METHOD PROTECTED OnStart
IF NOT Tco_TO_Tc2MC2_HomingMode(_homingMode, _mc_homingMode) THEN
    _message := Tc2_Standard.CONCAT('Unable to cast _homingMode variable of type TcoDrivesBeckhoff.eHomingMode (', TO_STRING(_homingMode));
    _message := Tc2_Standard.CONCAT(_message, ') to the type Tc2_MC2.MC_HomingMode!!!');
    THIS^.Messenger.Post(_message, TcoCore.eMessageCategory.ProgrammingError);
    ThrowWhen(TRUE);
    RETURN;
END_IF

IF NOT Tco_TO_Tc2MC2_Direction(_homingOptions_SearchDirection, _mc_homingOptions_SyncDirection) THEN
    _message := Tc2_Standard.CONCAT('Unable to cast _homingOptions_SearchDirection variable of type TcoDrivesBeckhoff.eDirection (',
        TO_STRING(_homingOptions_SearchDirection));

    _message := Tc2_Standard.CONCAT(_message, ') to the type Tc2_MC2.MC_Direction!!!');
    THIS^.Messenger.Post(_message, TcoCore.eMessageCategory.ProgrammingError);
    ThrowWhen(TRUE);
    RETURN;
END_IF

IF NOT Tco_TO_Tc2MC2_Direction(_homingOptions_SyncDirection, _mc_homingOptions_SyncDirection) THEN
    _message := Tc2_Standard.CONCAT('Unable to cast _homingOptions_SearchDirection variable of type TcoDrivesBeckhoff.eDirection (',
        TO_STRING(_homingOptions_SyncDirection));

    _message := Tc2_Standard.CONCAT(_message, ') to the type Tc2_MC2.MC_Direction!!!');
    THIS^.Messenger.Post(_message, TcoCore.eMessageCategory.ProgrammingError);
    ThrowWhen(TRUE);
    RETURN;
END_IF

IF NOT Tco_TO_Tc2MC2_EncRefMode(_homingOptions_ReferenceMode, _mc_homingOptions_ReferenceMode) THEN
    _message := Tc2_Standard.CONCAT('Unable to cast _homingOptions_ReferenceMode variable of type TcoDrivesBeckhoff.eEncoderReferenceMode (',
        TO_STRING(_homingOptions_ReferenceMode));

    _message := Tc2_Standard.CONCAT(_message, ') to the type Tc2_MC2.E_EncoderReferenceMode!!!');
    THIS^.Messenger.Post(_message, TcoCore.eMessageCategory.ProgrammingError);
    ThrowWhen(TRUE);
    RETURN;
END_IF

_mc_homingOptions.ClearPositionLag := _homingOptions_ClearPositionLag;
_mc_homingOptions.SearchDirection := _homingOptions_SearchDirection;
_mc_homingOptions.SearchVelocity := _homingOptions_SearchVelocity;
_mc_homingOptions.SyncDirection := _homingOptions_SyncDirection;
_mc_homingOptions.SyncVelocity := _homingOptions_SyncVelocity;
_mc_homingOptions.ReferenceMode := _homingOptions_ReferenceMode;
_calibrationCam := DriveRef.inCalibrationCam;
_mcHome(Axis := _axisRef, Execute := FALSE);
END_METHOD

(*~
    <docu>
        <summary>
            Restores this instance to the Ready state. Can be called explicitly or from within one of the restore mechanisms.
            <para>
                See also <see cref="PlcDocu.TcoCore.TcoTask.AutoRestorable()"/>
            </para>
        </summary>
    </docu>
~*)
METHOD Restore : ITcoRestorable
SUPER^.Restore();
END_METHOD

(*~
    <docu>
        <summary>
            Executes until task is in ```Error``` state .
        </summary>
    </docu>
~*)
METHOD PROTECTED WhileError
IF NOT _axisRef.Status.Error THEN
    DriveRef.SetErrorID(DriveRef._homeTask._mcHome.ErrorID);
    _mcHome(Axis := _axisRef, Execute := FALSE);
END_IF
END_METHOD

END_FUNCTION_BLOCK

// ---- POUs/Prototypes/TcoDriveSimple/Jog.TcPOU
FUNCTION_BLOCK Jog EXTENDS TcoCore.TcoObject IMPLEMENTS ITcoDriveSimple, TcoCore.ITcoServiceable
VAR_INPUT
    inIsServiceMode : BOOL;
END_VAR
VAR
    {attribute 'hide'}
    _axisRef : REFERENCE TO TcoAxisRef;
    {attribute 'hide'}
    _mcJog : Tc2_MC2.MC_Jog;
    {attribute addProperty Name "<#Jog forward#>"}
    {attribute addProperty StateOnDesc "<#Running#>"}
    {attribute addProperty StateOffDesc "<#Stopped#>"}
    _jogForwardTask : TcoCore.TcoMomentaryTask(THIS^);
    {attribute addProperty Name "<#Jog backwards#>"}
    {attribute addProperty StateOnDesc "<#Running#>"}
    {attribute addProperty StateOffDesc "<#Stopped#>"}
    _jogBackwardsTask : TcoCore.TcoMomentaryTask(THIS^);
    {attribute addProperty Name "<#Jog mode#>"}
    _jogMode : eJogMode;
    {attribute addProperty Name "<#Position#>"}
    _position : LREAL;
    {attribute addProperty Name "<#Velocity#>"}
    _velocity : LREAL;
    {attribute addProperty Name "<#Acceleration#>"}
    _acceleration : LREAL;
    {attribute addProperty Name "<#Deceleration#>"}
    _deceleration : LREAL;
    {attribute addProperty Name "<#Jerk#>"}
    _jerk : LREAL;
    {attribute 'hide'}
    _dummyPreconditionOK : BOOL;
    _serviceContexCycle : ULINT;
    _myContextCycleCount : ULINT;
    _inServiceMode : BOOL;
END_VAR

IF NOT __ISVALIDREF(_axisRef) THEN
    IF __ISVALIDREF(DriveRef) THEN
        _axisRef REF= DriveRef.AxisRef;
    ELSE
        RETURN;
    END_IF
END_IF

_jogForwardTask.Enabled := inIsServiceMode;
_jogBackwardsTask.Enabled := inIsServiceMode;
_jogForwardTask.Run();
_jogBackwardsTask.Run();

IF _jogForwardTask.State THEN
    _dummyPreconditionOK := DriveRef._power._mcPower.Enable_Positive;

    IF NOT DriveRef._movementState.JogPreconditionsOk(_jogForwardTask, _dummyPreconditionOK) THEN
        Messenger.Error('Movements to positive direction are disabled');
        RETURN;
    END_IF
END_IF

IF _jogBackwardsTask.State THEN
    _dummyPreconditionOK := DriveRef._power._mcPower.Enable_Negative;

    IF NOT DriveRef._movementState.JogPreconditionsOk(_jogBackwardsTask, _dummyPreconditionOK) THEN
        Messenger.Error('Movements to negative direction are disabled');
        RETURN;
    END_IF
END_IF

_mcJog(Axis := _axisRef,
    JogForward := _jogForwardTask.State AND NOT _mcJog.Error,
    JogBackwards := _jogBackwardsTask.State AND NOT _mcJog.Error,
    Mode := _jogMode,
    Position := _position,
    Velocity := _velocity,
    Acceleration := _acceleration,
    Deceleration := _deceleration,
    Jerk := _jerk,
    Done =>,
    Busy =>,
    Active =>,
    CommandAborted =>,
    Error =>,
    ErrorID =>);

IF _mcJog.Done OR _mcJog.CommandAborted OR _mcJog.Error THEN
    THIS^.DriveRef._movementState.Restore();
END_IF

IF NOT _axisRef.Status.Error AND _mcJog.Error THEN
    DriveRef.SetErrorID(_mcJog.ErrorID);
END_IF

PROPERTY DriveRef : REFERENCE TO TcoDriveSimple
GET
VAR
    _drive : ITcoDriveSimple := 0;
END_VAR
IF __QUERYINTERFACE(THIS^.Parent, _drive) THEN
    DriveRef REF= _drive.DriveRef;
END_IF
END_GET
END_PROPERTY

METHOD FB_init : BOOL
VAR_INPUT
    bInitRetains : BOOL; // if TRUE, the retain variables are initialized (warm start / cold start)
    bInCopyCode : BOOL; // if TRUE, the instance afterwards gets moved into the copy code (online change)
    ParentObject : ITcoObject;
END_VAR
END_METHOD

PROPERTY IsService : BOOL
GET
_myContextCycleCount := Context.StartCycleCount;
//When component.Service() is called "before" invoking its task _serviceContexCycle is equal to Context.StartCycleCount
//When component.Service() is called "after" invoking its task (_serviceContexCycle + 1) is equal to Context.StartCycleCount
//otherwise _serviceContexCycle should be lower then Context.StartCycleCount until Context.StartCycleCount overflow its range
//which should occur cca every 585 mil years at 1ms PLC task.
_inServiceMode := _serviceContexCycle = _myContextCycleCount OR (_serviceContexCycle + 1) = _myContextCycleCount;
IsService := _inServiceMode;
END_GET
END_PROPERTY

METHOD PUBLIC Service
_serviceContexCycle := Context.StartCycleCount;
END_METHOD

END_FUNCTION_BLOCK

// ---- POUs/Prototypes/TcoDriveSimple/MotionTasks/SetTorqueTask.TcPOU
FUNCTION_BLOCK SetTorqueTask EXTENDS TcoCore.TcoTask IMPLEMENTS ITcoDriveSimple
VAR_INPUT
    inIsServiceMode : BOOL;
END_VAR
VAR
    {attribute addProperty Name "<#Torque/Force#>"}
    _torque : LREAL;
    {attribute addProperty Name "<#Relative#>"}
    _relative : BOOL;
    {attribute addProperty Name "<#Velocity limit high#>"}
    _velocityLimitHigh : LREAL;
    {attribute addProperty Name "<#Velocity limit low#>"}
    _velocityLimitLow : LREAL;
    {attribute addProperty Name "<#Continuous update#>"}
    _continuousUpdate : BOOL := TRUE;
    {attribute addProperty Name "<#Torque ramp#>"}
    _torqueRamp : LREAL;
    {attribute addProperty Name "<#Torque Options: Enable Manual Torque Start value #>"}
    _enableManualTorqueStartValue : BOOL;
    {attribute addProperty Name "<#Torque Options:Manual Torque Start value#>"}
    _manualTorqueStartValue : LREAL;
END_VAR
VAR
    {attribute 'hide'}
    _axisRef : REFERENCE TO TcoAxisRef;
    {attribute 'hide'}
    _mcTorqueControl : Tc2_MC2.MC_TorqueControl;
    {attribute 'hide'}
    _torqueOptions : Tc2_MC2.ST_TorqueControlOptions;
    {attribute 'hide'}
    _message : STRING(125);
END_VAR

IF NOT __ISVALIDREF(_axisRef) THEN
    IF __ISVALIDREF(DriveRef) THEN
        _axisRef REF= DriveRef.AxisRef;
    ELSE
        RETURN;
    END_IF
END_IF

IF Execute() THEN
    IF inIsServiceMode AND _enableManualTorqueStartValue THEN
        _torqueOptions.EnableManualTorqueStartValue := _enableManualTorqueStartValue;
        _torqueOptions.ManualTorqueStartValue := _manualTorqueStartValue;
    END_IF;

    _mcTorqueControl(Axis := _axisRef,
        Execute := NOT _mcTorqueControl.Busy,
        ContinuousUpdate := _continuousUpdate,
        Relative := _relative,
        Torque := _torque,
        TorqueRamp := _torqueRamp,
        VelocityLimitHigh := _velocityLimitHigh,
        VelocityLimitLow := _velocityLimitLow,
        BufferMode := Tc2_MC2.MC_Aborting,
        Options := _torqueOptions,
        InTorque =>,
        Busy =>,
        Active =>,
        CommandAborted =>,
        Error =>,
        ErrorId =>);

    IF _mcTorqueControl.CommandAborted THEN
        THIS^.Abort();
    END_IF

    DoneWhen(_mcTorqueControl.InTorque);
    ThrowWhen(_mcTorqueControl.Error);
END_IF

PROPERTY DriveRef : REFERENCE TO TcoDriveSimple
GET
VAR
    _drive : ITcoDriveSimple := 0;
END_VAR
IF __QUERYINTERFACE(THIS^.Parent, _drive) THEN
    DriveRef REF= _drive.DriveRef;
END_IF
END_GET
END_PROPERTY

PROPERTY PUBLIC InTorque : BOOL
GET
InTorque := _mcTorqueControl.InTorque;
END_GET
END_PROPERTY

METHOD INTERNAL InvokeWithParams : ITcoTaskStatus
VAR_INPUT
    inTorque : LREAL;
    inRelative : BOOL;
    inVelocityLimitHigh : LREAL;
    inVelocityLimitLow : LREAL;
    inContinuousUpdate : BOOL := TRUE;
    inTorqueRamp : LREAL;
    inTorqueOptions : Tc2_MC2.ST_TorqueControlOptions;
END_VAR
_torque := inTorque;
_relative := inRelative;
_velocityLimitHigh := inVelocityLimitHigh;
_velocityLimitLow := inVelocityLimitLow;
_continuousUpdate := inContinuousUpdate;
_torqueRamp := inTorqueRamp;
_torqueOptions := inTorqueOptions;
InvokeWithParams := THIS^.Invoke();
END_METHOD

(*~
    <docu>
        <summary>
            Executes when task is aborted.
        </summary>
    </docu>
~*)
METHOD PROTECTED OnAbort
IF NOT __ISVALIDREF(_axisRef) THEN
    IF __ISVALIDREF(DriveRef) THEN
        _axisRef REF= DriveRef.AxisRef;
    ELSE
        RETURN;
    END_IF
END_IF

THIS^.DriveRef.Stop(-1, -1);
_mcTorqueControl(Axis := _axisRef, Execute := FALSE);
THIS^.DriveRef._movementState.Restore();
END_METHOD

(*~
    <docu>
        <summary>
            Executes when task reaches the ```Done``` state .
        </summary>
    </docu>
~*)
METHOD PROTECTED OnDone
_mcTorqueControl(Axis := _axisRef, Execute := FALSE);
THIS^.DriveRef._movementState.Restore();
END_METHOD

(*~
    <docu>
        <summary>
            Executes when task reaches the ```Error``` state.
            <para>
                Do not confuse with <see cref="PlcDocu.TcoCore.TcoTask.WhileError()"/>, that is called cyclically until '''Error''' state is left.
            </para>
        </summary>
    </docu>
~*)
METHOD PROTECTED OnError
THIS^.DriveRef._movementState.Restore();

IF NOT _axisRef.Status.Error THEN
    DriveRef.SetErrorID(DriveRef._axisStatus.ErrorId);
END_IF

_mcTorqueControl(Axis := _axisRef, Execute := FALSE);
END_METHOD

METHOD PROTECTED OnStart
_mcTorqueControl(Axis := _axisRef, Execute := FALSE);
END_METHOD

(*~
    <docu>
        <summary>
            Restores this instance to the Ready state. Can be called explicitly or from within one of the restore mechanisms.
            <para>
                See also <see cref="PlcDocu.TcoCore.TcoTask.AutoRestorable()"/>
            </para>
        </summary>
    </docu>
~*)
METHOD Restore : ITcoRestorable
SUPER^.Restore();
END_METHOD

(*~
    <docu>
        <summary>
            Executes until task is in ```Error``` state .
            <para>
                Do not confuse with <see cref="PlcDocu.TcoCore.TcoTask.OnError()"/>, that is called just ones when '''Error''' state is entered.
            </para>
        </summary>
    </docu>
~*)
METHOD PROTECTED WhileError
IF NOT _axisRef.Status.Error THEN
    DriveRef.SetErrorID(_mcTorqueControl.ErrorID);
    _mcTorqueControl(Axis := _axisRef, Execute := FALSE);
END_IF
END_METHOD

END_FUNCTION_BLOCK

// ---- POUs/Prototypes/TcoDriveSimple/MotionTasks/MoveVelocityTask.TcPOU
FUNCTION_BLOCK MoveVelocityTask EXTENDS TcoCore.TcoTask IMPLEMENTS ITcoDriveSimple
VAR
    {attribute addProperty Name "<#Velocity#>"}
    _velocity : LREAL;
    {attribute addProperty Name "<#Acceleration#>"}
    _acceleration : LREAL;
    {attribute addProperty Name "<#Deceleration#>"}
    _deceleration : LREAL;
    {attribute addProperty Name "<#Jerk#>"}
    _jerk : LREAL;
    {attribute addProperty Name "<#Direction#>"}
    _direction : eDirection;
END_VAR
VAR
    {attribute 'hide'}
    _axisRef : REFERENCE TO TcoAxisRef;
    {attribute 'hide'}
    _mcMoveVelocity : Tc2_MC2.MC_MoveVelocity;
    {attribute 'hide'}
    _mc_direction : Tc2_MC2.MC_Direction;
    {attribute 'hide'}
    _message : STRING(125);
    {attribute 'hide'}
    _dummyPreconditionOK : BOOL;
END_VAR

IF NOT __ISVALIDREF(_axisRef) THEN
    IF __ISVALIDREF(DriveRef) THEN
        _axisRef REF= DriveRef.AxisRef;
    ELSE
        RETURN;
    END_IF
END_IF

IF Execute() THEN
    _dummyPreconditionOK := TRUE;

    IF NOT DriveRef._movementState.MovePreconditionsOk(THIS^, _dummyPreconditionOK) THEN
        Messenger.Error('To be implemented');
        RETURN;
    END_IF

    _mcMoveVelocity(Axis := _axisRef,
        Execute := NOT _mcMoveVelocity.Busy,
        Velocity := _velocity,
        Acceleration := _acceleration,
        Deceleration := _deceleration,
        Jerk := _jerk,
        Direction := _mc_direction,
        BufferMode := Tc2_MC2.MC_Aborting,
        InVelocity =>,
        Busy =>,
        Active =>,
        CommandAborted =>,
        Error =>,
        ErrorID =>);

    IF _mcMoveVelocity.CommandAborted THEN
        THIS^.Abort();
    END_IF

    DoneWhen(_mcMoveVelocity.InVelocity);
    ThrowWhen(_mcMoveVelocity.Error);
END_IF

PROPERTY DriveRef : REFERENCE TO TcoDriveSimple
GET
VAR
    _drive : ITcoDriveSimple := 0;
END_VAR
IF __QUERYINTERFACE(THIS^.Parent, _drive) THEN
    DriveRef REF= _drive.DriveRef;
END_IF
END_GET
END_PROPERTY

METHOD PUBLIC FB_init : BOOL
VAR_INPUT
    bInitRetains : BOOL; // if TRUE, the retain variables are initialized (warm start / cold start)
    bInCopyCode : BOOL; // if TRUE, the instance afterwards gets moved into the copy code (online change)
    ParentObject : ITcoObject;
END_VAR
END_METHOD

PROPERTY PUBLIC InVelocity : BOOL
GET
InVelocity := _mcMoveVelocity.InVelocity;
END_GET
END_PROPERTY

METHOD INTERNAL InvokeWithParams : ITcoTaskStatus
VAR_INPUT
    inVelocity : LREAL;
    inAcceleration : LREAL;
    inDeceleration : LREAL;
    inJerk : LREAL;
    inDirection : eDirection;
END_VAR
_velocity := inVelocity;
_acceleration := inAcceleration;
_deceleration := inDeceleration;
_jerk := inJerk;
_direction := inDirection;
InvokeWithParams := THIS^.Invoke();
END_METHOD

(*~
    <docu>
        <summary>
            Executes when task is aborted.
        </summary>
    </docu>
~*)
METHOD PROTECTED OnAbort
IF NOT __ISVALIDREF(_axisRef) THEN
    IF __ISVALIDREF(DriveRef) THEN
        _axisRef REF= DriveRef.AxisRef;
    ELSE
        RETURN;
    END_IF
END_IF

THIS^.DriveRef.Stop(-1, -1);
THIS^.DriveRef._movementState.Restore();
_mcMoveVelocity(Axis := _axisRef, Execute := FALSE);
END_METHOD

(*~
    <docu>
        <summary>
            Executes when task reaches the ```Done``` state .
        </summary>
    </docu>
~*)
METHOD PROTECTED OnDone
THIS^.DriveRef._movementState.Restore();
_mcMoveVelocity(Axis := _axisRef, Execute := FALSE);
END_METHOD

(*~
    <docu>
        <summary>
            Executes when task reaches the ```Error``` state.
            <para>
                Do not confuse with <see cref="PlcDocu.TcoCore.TcoTask.WhileError()"/>, that is called cyclically until '''Error''' state is left.
            </para>
        </summary>
    </docu>
~*)
METHOD PROTECTED OnError
THIS^.DriveRef._movementState.Restore();

IF NOT _axisRef.Status.Error THEN
    DriveRef.SetErrorID(DriveRef._moveVelocityTask._mcMoveVelocity.ErrorID);
END_IF

_mcMoveVelocity(Axis := _axisRef, Execute := FALSE);
END_METHOD

METHOD PROTECTED OnStart
IF NOT Tco_TO_Tc2MC2_Direction(_direction, _mc_direction) THEN
    _message := Tc2_Standard.CONCAT('Unable to cast _direction variable of type TcoDrivesBeckhoff.eDirection (', TO_STRING(_direction));
    _message := Tc2_Standard.CONCAT(_message, ') to the type Tc2_MC2.MC_Direction!!!');
    THIS^.Messenger.Post(_message, TcoCore.eMessageCategory.ProgrammingError);
    ThrowWhen(TRUE);
    RETURN;
END_IF

_mcMoveVelocity(Axis := _axisRef, Execute := FALSE);
END_METHOD

(*~
    <docu>
        <summary>
            Restores this instance to the Ready state. Can be called explicitly or from within one of the restore mechanisms.
            <para>
                See also <see cref="PlcDocu.TcoCore.TcoTask.AutoRestorable()"/>
            </para>
        </summary>
    </docu>
~*)
METHOD Restore : ITcoRestorable
SUPER^.Restore();
END_METHOD

(*~
    <docu>
        <summary>
            Executes until task is in ```Error``` state .
        </summary>
    </docu>
~*)
METHOD PROTECTED WhileError
IF NOT _axisRef.Status.Error THEN
    DriveRef.SetErrorID(DriveRef._moveVelocityTask._mcMoveVelocity.ErrorID);
    _mcMoveVelocity(Axis := _axisRef, Execute := FALSE);
END_IF
END_METHOD

END_FUNCTION_BLOCK

// ---- POUs/Prototypes/TcoDriveSimple/MotionTasks/StopTask.TcPOU
FUNCTION_BLOCK StopTask EXTENDS TcoCore.TcoTask IMPLEMENTS ITcoDriveSimple
VAR
    {attribute addProperty Name "<#Deceleration#>"}
    _deceleration : LREAL;
    {attribute addProperty Name "<#Jerk#>"}
    _jerk : LREAL;
END_VAR
VAR
    {attribute 'hide'}
    _axisRef : REFERENCE TO TcoAxisRef;
    {attribute 'hide'}
    _mcStop : Tc2_MC2.MC_Stop;
END_VAR

IF NOT __ISVALIDREF(_axisRef) THEN
    IF __ISVALIDREF(DriveRef) THEN
        _axisRef REF= DriveRef.AxisRef;
    ELSE
        RETURN;
    END_IF
END_IF

_mcStop(Axis := _axisRef, Execute := FALSE);

IF Execute() THEN
    _mcStop(Axis := _axisRef,
        Execute := NOT _mcStop.Busy,
        Deceleration := _deceleration,
        Jerk := _jerk,
        Done =>,
        Busy =>,
        Active =>,
        CommandAborted =>,
        Error =>,
        ErrorID =>);

    IF _mcStop.CommandAborted THEN
        THIS^.Abort();
    END_IF

    DoneWhen(_mcStop.Done);
    ThrowWhen(_mcStop.Error);
END_IF

PROPERTY DriveRef : REFERENCE TO TcoDriveSimple
GET
VAR
    _drive : ITcoDriveSimple := 0;
END_VAR
IF __QUERYINTERFACE(THIS^.Parent, _drive) THEN
    DriveRef REF= _drive.DriveRef;
END_IF
END_GET
END_PROPERTY

METHOD PUBLIC FB_init : BOOL
VAR_INPUT
    bInitRetains : BOOL; // if TRUE, the retain variables are initialized (warm start / cold start)
    bInCopyCode : BOOL; // if TRUE, the instance afterwards gets moved into the copy code (online change)
    ParentObject : ITcoObject;
END_VAR
END_METHOD

METHOD INTERNAL InvokeWithParams : ITcoTaskStatus
VAR_INPUT
    inDeceleration : LREAL;
    inJerk : LREAL;
END_VAR
_deceleration := inDeceleration;
_jerk := inJerk;
InvokeWithParams := THIS^.Invoke();
END_METHOD

(*~
    <docu>
        <summary>
            Executes when task is aborted.
        </summary>
    </docu>
~*)
METHOD PROTECTED OnAbort
THIS^.DriveRef._movementState.Restore();
_mcStop(Axis := _axisRef, Execute := FALSE);
END_METHOD

(*~
    <docu>
        <summary>
            Executes when task reaches the ```Done``` state .
        </summary>
    </docu>
~*)
METHOD PROTECTED OnDone
THIS^.DriveRef._movementState.Restore();
_mcStop(Axis := _axisRef, Execute := FALSE);
END_METHOD

(*~
    <docu>
        <summary>
            Executes when task reaches the ```Error``` state.
            <para>
                Do not confuse with <see cref="PlcDocu.TcoCore.TcoTask.WhileError()"/>, that is called cyclically until '''Error''' state is left.
            </para>
        </summary>
    </docu>
~*)
METHOD PROTECTED OnError
THIS^.DriveRef._movementState.Restore();

IF NOT _axisRef.Status.Error THEN
    DriveRef.SetErrorID(DriveRef._stopTask._mcStop.ErrorID);
END_IF

_mcStop(Axis := _axisRef, Execute := FALSE);
END_METHOD

METHOD PROTECTED OnStart
_mcStop(Axis := _axisRef, Execute := FALSE);
END_METHOD

(*~
    <docu>
        <summary>
            Restores this instance to the Ready state. Can be called explicitly or from within one of the restore mechanisms.
            <para>
                See also <see cref="PlcDocu.TcoCore.TcoTask.AutoRestorable()"/>
            </para>
        </summary>
    </docu>
~*)
METHOD Restore : ITcoRestorable
SUPER^.Restore();
END_METHOD

(*~
    <docu>
        <summary>
            Executes until task is in ```Error``` state .
        </summary>
    </docu>
~*)
METHOD PROTECTED WhileError
IF NOT _axisRef.Status.Error THEN
    DriveRef.SetErrorID(DriveRef._stopTask._mcStop.ErrorID);
    _mcStop(Axis := _axisRef, Execute := FALSE);
END_IF
END_METHOD

END_FUNCTION_BLOCK

// ---- POUs/Prototypes/TcoDriveSimple/MotionTasks/HaltTask.TcPOU
FUNCTION_BLOCK HaltTask EXTENDS TcoCore.TcoTask IMPLEMENTS ITcoDriveSimple
VAR
    {attribute addProperty Name "<#Deceleration#>"}
    _deceleration : LREAL;
    {attribute addProperty Name "<#Jerk#>"}
    _jerk : LREAL;
END_VAR
VAR
    {attribute 'hide'}
    _axisRef : REFERENCE TO TcoAxisRef;
    {attribute 'hide'}
    _mcHalt : Tc2_MC2.MC_Halt;
END_VAR

IF NOT __ISVALIDREF(_axisRef) THEN
    IF __ISVALIDREF(DriveRef) THEN
        _axisRef REF= DriveRef.AxisRef;
    ELSE
        RETURN;
    END_IF
END_IF

IF Execute() THEN
    _mcHalt(Axis := _axisRef);

    IF _mcHalt.CommandAborted THEN
        THIS^.Abort();
    END_IF

    DoneWhen(_mcHalt.Done);
    ThrowWhen(_mcHalt.Error);
END_IF

PROPERTY DriveRef : REFERENCE TO TcoDriveSimple
GET
VAR
    _drive : ITcoDriveSimple := 0;
END_VAR
IF __QUERYINTERFACE(THIS^.Parent, _drive) THEN
    DriveRef REF= _drive.DriveRef;
END_IF
END_GET
END_PROPERTY

METHOD PUBLIC FB_init : BOOL
VAR_INPUT
    bInitRetains : BOOL; // if TRUE, the retain variables are initialized (warm start / cold start)
    bInCopyCode : BOOL; // if TRUE, the instance afterwards gets moved into the copy code (online change)
    ParentObject : ITcoObject;
END_VAR
END_METHOD

METHOD INTERNAL InvokeWithParams : ITcoTaskStatus
VAR_INPUT
    inDeceleration : LREAL;
    inJerk : LREAL;
END_VAR
_deceleration := inDeceleration;
_jerk := inJerk;
InvokeWithParams := THIS^.Invoke();
END_METHOD

(*~
    <docu>
        <summary>
            Executes when task is aborted.
        </summary>
    </docu>
~*)
METHOD PROTECTED OnAbort
_mcHalt(Axis := _axisRef, Execute := FALSE, Deceleration := _deceleration);
THIS^.DriveRef._movementState.Restore();
END_METHOD

(*~
    <docu>
        <summary>
            Executes when task reaches the ```Done``` state .
        </summary>
    </docu>
~*)
METHOD PROTECTED OnDone
_mcHalt(Axis := _axisRef, Execute := FALSE, Deceleration := _deceleration);
THIS^.DriveRef._movementState.Restore();
END_METHOD

(*~
    <docu>
        <summary>
            Executes when task reaches the ```Error``` state.
            <para>
                Do not confuse with <see cref="PlcDocu.TcoCore.TcoTask.WhileError()"/>, that is called cyclically until '''Error''' state is left.
            </para>
        </summary>
    </docu>
~*)
METHOD PROTECTED OnError
THIS^.DriveRef._movementState.Restore();

IF NOT _axisRef.Status.Error THEN
    DriveRef.SetErrorID(DriveRef._haltTask._mcHalt.ErrorID);
END_IF

_mcHalt(Axis := _axisRef, Execute := FALSE);
END_METHOD

METHOD PROTECTED OnStart
_mcHalt(Axis := _axisRef, Execute := false, Deceleration := _deceleration);
_mcHalt(Axis := _axisRef, Execute := TRUE, Deceleration := _deceleration);
END_METHOD

(*~
    <docu>
        <summary>
            Restores this instance to the Ready state. Can be called explicitly or from within one of the restore mechanisms.
            <para>
                See also <see cref="PlcDocu.TcoCore.TcoTask.AutoRestorable()"/>
            </para>
        </summary>
    </docu>
~*)
METHOD Restore : ITcoRestorable
SUPER^.Restore();
END_METHOD

(*~
    <docu>
        <summary>
            Executes until task is in ```Error``` state .
        </summary>
    </docu>
~*)
METHOD PROTECTED WhileError
IF NOT _axisRef.Status.Error THEN
    DriveRef.SetErrorID(DriveRef._haltTask._mcHalt.ErrorID);
    _mcHalt(Axis := _axisRef, Execute := FALSE);
END_IF
END_METHOD

END_FUNCTION_BLOCK

// ---- POUs/Prototypes/TcoDriveSimple/MotionTasks/MoveRelativeTask.TcPOU
FUNCTION_BLOCK MoveRelativeTask EXTENDS TcoCore.TcoTask IMPLEMENTS ITcoDriveSimple
VAR
    {attribute addProperty Name "<#Distance#>"}
    _distance : LREAL;
    {attribute addProperty Name "<#Velocity#>"}
    _velocity : LREAL;
    {attribute addProperty Name "<#Acceleration#>"}
    _acceleration : LREAL;
    {attribute addProperty Name "<#Deceleration#>"}
    _deceleration : LREAL;
    {attribute addProperty Name "<#Jerk#>"}
    _jerk : LREAL;
END_VAR
VAR
    {attribute 'hide'}
    _axisRef : REFERENCE TO TcoAxisRef;
    {attribute 'hide'}
    _mcMoveRelative : Tc2_MC2.MC_MoveRelative;
    {attribute 'hide'}
    _dummyPreconditionOK : BOOL;
END_VAR

IF NOT __ISVALIDREF(_axisRef) THEN
    IF __ISVALIDREF(DriveRef) THEN
        _axisRef REF= DriveRef.AxisRef;
    ELSE
        RETURN;
    END_IF
END_IF

IF Execute() THEN
    _dummyPreconditionOK := TRUE;

    IF NOT DriveRef._movementState.MovePreconditionsOk(THIS^, _dummyPreconditionOK) THEN
        Messenger.Error('To be implemented');
        RETURN;
    END_IF

    _mcMoveRelative(Axis := _axisRef,
        Execute := NOT _mcMoveRelative.Busy,
        Distance := _distance,
        Velocity := _velocity,
        Acceleration := _acceleration,
        Deceleration := _deceleration,
        Jerk := _jerk,
        BufferMode := Tc2_MC2.MC_Aborting,
        Done =>,
        Busy =>,
        Active =>,
        CommandAborted =>,
        Error =>,
        ErrorID =>);

    IF _mcMoveRelative.CommandAborted THEN
        THIS^.Abort();
    END_IF

    DoneWhen(_mcMoveRelative.Done);
    ThrowWhen(_mcMoveRelative.Error);
END_IF

PROPERTY DriveRef : REFERENCE TO TcoDriveSimple
GET
VAR
    _drive : ITcoDriveSimple := 0;
END_VAR
IF __QUERYINTERFACE(THIS^.Parent, _drive) THEN
    DriveRef REF= _drive.DriveRef;
END_IF
END_GET
END_PROPERTY

METHOD PUBLIC FB_init : BOOL
VAR_INPUT
    bInitRetains : BOOL; // if TRUE, the retain variables are initialized (warm start / cold start)
    bInCopyCode : BOOL; // if TRUE, the instance afterwards gets moved into the copy code (online change)
    ParentObject : ITcoObject;
END_VAR
END_METHOD

METHOD INTERNAL InvokeWithParams : ITcoTaskStatus
VAR_INPUT
    inDistance : LREAL;
    inVelocity : LREAL;
    inAcceleration : LREAL;
    inDeceleration : LREAL;
    inJerk : LREAL;
END_VAR
_distance := inDistance;
_velocity := inVelocity;
_acceleration := inAcceleration;
_deceleration := inDeceleration;
_jerk := inJerk;
InvokeWithParams := THIS^.Invoke();
END_METHOD

(*~
    <docu>
        <summary>
            Executes when task is aborted.
        </summary>
    </docu>
~*)
METHOD PROTECTED OnAbort
IF NOT __ISVALIDREF(_axisRef) THEN
    IF __ISVALIDREF(DriveRef) THEN
        _axisRef REF= DriveRef.AxisRef;
    ELSE
        RETURN;
    END_IF
END_IF

THIS^.DriveRef.Stop(-1, -1);
THIS^.DriveRef._movementState.Restore();
_mcMoveRelative(Axis := _axisRef, Execute := FALSE);
END_METHOD

(*~
    <docu>
        <summary>
            Executes when task reaches the ```Done``` state .
        </summary>
    </docu>
~*)
METHOD PROTECTED OnDone
THIS^.DriveRef._movementState.Restore();
_mcMoveRelative(Axis := _axisRef, Execute := FALSE);
END_METHOD

(*~
    <docu>
        <summary>
            Executes when task reaches the ```Error``` state.
            <para>
                Do not confuse with <see cref="PlcDocu.TcoCore.TcoTask.WhileError()"/>, that is called cyclically until '''Error''' state is left.
            </para>
        </summary>
    </docu>
~*)
METHOD PROTECTED OnError
THIS^.DriveRef._movementState.Restore();

IF NOT _axisRef.Status.Error THEN
    DriveRef.SetErrorID(DriveRef._moveRelativeTask._mcMoveRelative.ErrorID);
END_IF

_mcMoveRelative(Axis := _axisRef, Execute := FALSE);
END_METHOD

METHOD PROTECTED OnStart
_mcMoveRelative(Axis := _axisRef, Execute := FALSE);
END_METHOD

(*~
    <docu>
        <summary>
            Restores this instance to the Ready state. Can be called explicitly or from within one of the restore mechanisms.
            <para>
                See also <see cref="PlcDocu.TcoCore.TcoTask.AutoRestorable()"/>
            </para>
        </summary>
    </docu>
~*)
METHOD Restore : ITcoRestorable
SUPER^.Restore();
END_METHOD

(*~
    <docu>
        <summary>
            Executes until task is in ```Error``` state .
        </summary>
    </docu>
~*)
METHOD PROTECTED WhileError
IF NOT _axisRef.Status.Error THEN
    DriveRef.SetErrorID(DriveRef._moveRelativeTask._mcMoveRelative.ErrorID);
    _mcMoveRelative(Axis := _axisRef, Execute := FALSE);
END_IF
END_METHOD

END_FUNCTION_BLOCK

// ---- POUs/Prototypes/TcoDriveSimple/MotionTasks/MoveAbsoluteTask.TcPOU
FUNCTION_BLOCK MoveAbsoluteTask EXTENDS TcoCore.TcoTask IMPLEMENTS ITcoDriveSimple
VAR
    {attribute addProperty Name "<#Position#>"}
    _position : LREAL;
    {attribute addProperty Name "<#Velocity#>"}
    _velocity : LREAL;
    {attribute addProperty Name "<#Acceleration#>"}
    _acceleration : LREAL;
    {attribute addProperty Name "<#Deceleration#>"}
    _deceleration : LREAL;
    {attribute addProperty Name "<#Jerk#>"}
    _jerk : LREAL;
END_VAR
VAR
    {attribute 'hide'}
    _axisRef : REFERENCE TO TcoAxisRef;
    {attribute 'hide'}
    _mcMoveAbsolute : Tc2_MC2.MC_MoveAbsolute;
    {attribute 'hide'}
    _mcMoveAbsolutePreconditionOK : BOOL;
    {attribute 'hide'}
    _mcReadAxisEncoderReferenceSystem : MC_ReadParameter;
    _AxisEncoderReferenceSystem : eAxisEncoderReferenceSystem;
END_VAR

IF NOT __ISVALIDREF(_axisRef) THEN
    IF __ISVALIDREF(DriveRef) THEN
        _axisRef REF= DriveRef.AxisRef;
    ELSE
        RETURN;
    END_IF
END_IF

IF Execute() THEN
    _mcReadAxisEncoderReferenceSystem(Axis := _axisRef,
        Enable := TRUE,
        ParameterNumber := eAxisParameter.AxisEncoderReferenceSystem,
        ReadMode := Tc2_MC2.E_ReadMode.READMODE_ONCE);

    IF _mcReadAxisEncoderReferenceSystem.Valid THEN
        LREAL_TO_Tco_AxisEncoderReferenceSystem(_mcReadAxisEncoderReferenceSystem.Value, _AxisEncoderReferenceSystem);

        IF _AxisEncoderReferenceSystem = eAxisEncoderReferenceSystem.ABSOLUTE OR
            _AxisEncoderReferenceSystem = eAxisEncoderReferenceSystem.ABSOLUTE_MODULO OR
            _AxisEncoderReferenceSystem = eAxisEncoderReferenceSystem.ABSOLUTE_MULTITURN OR
            _AxisEncoderReferenceSystem = eAxisEncoderReferenceSystem.ABSOLUTE_SINGLETURN THEN
            _mcMoveAbsolutePreconditionOK := TRUE;
        ELSE
            _mcMoveAbsolutePreconditionOK := _axisRef.Status.Homed;
        END_IF
    END_IF

    IF NOT DriveRef._movementState.MovePreconditionsOk(THIS^, _mcMoveAbsolutePreconditionOK) THEN
        IF _mcReadAxisEncoderReferenceSystem.Valid AND NOT _mcMoveAbsolutePreconditionOK THEN
            Messenger.Error('Move absolute not possible as axis is Incremental and not Homed');
        END_IF

        RETURN;
    END_IF

    _mcMoveAbsolute(Axis := _axisRef,
        Execute := NOT _mcMoveAbsolute.Busy,
        Position := _position,
        Velocity := _velocity,
        Acceleration := _acceleration,
        Deceleration := _deceleration,
        Jerk := _jerk,
        BufferMode := Tc2_MC2.MC_Aborting,
        Done =>,
        Busy =>,
        Active =>,
        CommandAborted =>,
        Error =>,
        ErrorID =>);

    IF _mcMoveAbsolute.CommandAborted THEN
        THIS^.Abort();
    END_IF

    DoneWhen(_mcMoveAbsolute.Done);
    ThrowWhen(_mcMoveAbsolute.Error);
END_IF

PROPERTY DriveRef : REFERENCE TO TcoDriveSimple
GET
VAR
    _drive : ITcoDriveSimple := 0;
END_VAR
IF __QUERYINTERFACE(THIS^.Parent, _drive) THEN
    DriveRef REF= _drive.DriveRef;
END_IF
END_GET
END_PROPERTY

METHOD PUBLIC FB_init : BOOL
VAR_INPUT
    bInitRetains : BOOL; // if TRUE, the retain variables are initialized (warm start / cold start)
    bInCopyCode : BOOL; // if TRUE, the instance afterwards gets moved into the copy code (online change)
    ParentObject : ITcoObject;
END_VAR
END_METHOD

METHOD INTERNAL InvokeWithParams : ITcoTaskStatus
VAR_INPUT
    inPosition : LREAL;
    inVelocity : LREAL;
    inAcceleration : LREAL;
    inDeceleration : LREAL;
    inJerk : LREAL;
END_VAR
_position := inPosition;
_velocity := inVelocity;
_acceleration := inAcceleration;
_deceleration := inDeceleration;
_jerk := inJerk;
InvokeWithParams := THIS^.Invoke();
END_METHOD

(*~
    <docu>
        <summary>
            Executes when task is aborted.
        </summary>
    </docu>
~*)
METHOD PROTECTED OnAbort
IF NOT __ISVALIDREF(_axisRef) THEN
    IF __ISVALIDREF(DriveRef) THEN
        _axisRef REF= DriveRef.AxisRef;
    ELSE
        RETURN;
    END_IF
END_IF

THIS^.DriveRef.Stop(-1, -1);
_mcMoveAbsolute(Axis := _axisRef, Execute := FALSE);
_mcReadAxisEncoderReferenceSystem(Axis := _axisRef, Enable := FALSE);
THIS^.DriveRef._movementState.Restore();
END_METHOD

(*~
    <docu>
        <summary>
            Executes when task reaches the ```Done``` state .
        </summary>
    </docu>
~*)
METHOD PROTECTED OnDone
_mcMoveAbsolute(Axis := _axisRef, Execute := FALSE);
_mcReadAxisEncoderReferenceSystem(Axis := _axisRef, Enable := FALSE);
THIS^.DriveRef._movementState.Restore();
END_METHOD

(*~
    <docu>
        <summary>
            Executes when task reaches the ```Error``` state.
            <para>
                Do not confuse with <see cref="PlcDocu.TcoCore.TcoTask.WhileError()"/>, that is called cyclically until '''Error''' state is left.
            </para>
        </summary>
    </docu>
~*)
METHOD PROTECTED OnError
THIS^.DriveRef._movementState.Restore();

IF NOT _axisRef.Status.Error THEN
    DriveRef.SetErrorID(DriveRef._moveAbsoluteTask._mcMoveAbsolute.ErrorID);
END_IF

_mcMoveAbsolute(Axis := _axisRef, Execute := FALSE);
_mcReadAxisEncoderReferenceSystem(Axis := _axisRef, Enable := FALSE);
END_METHOD

METHOD PROTECTED OnStart
_mcMoveAbsolute(Axis := _axisRef, Execute := FALSE);
_mcReadAxisEncoderReferenceSystem(Axis := _axisRef, Enable := FALSE);
END_METHOD

(*~
    <docu>
        <summary>
            Restores this instance to the Ready state. Can be called explicitly or from within one of the restore mechanisms.
            <para>
                See also <see cref="PlcDocu.TcoCore.TcoTask.AutoRestorable()"/>
            </para>
        </summary>
    </docu>
~*)
METHOD Restore : ITcoRestorable
SUPER^.Restore();
END_METHOD

(*~
    <docu>
        <summary>
            Executes until task is in ```Error``` state .
        </summary>
    </docu>
~*)
METHOD PROTECTED WhileError
IF NOT _axisRef.Status.Error THEN
    DriveRef.SetErrorID(DriveRef._moveAbsoluteTask._mcMoveAbsolute.ErrorID);
    _mcMoveAbsolute(Axis := _axisRef, Execute := FALSE);
END_IF
END_METHOD

END_FUNCTION_BLOCK

// ---- POUs/Prototypes/TcoDriveSimple/MotionTasks/MoveModuloTask.TcPOU
FUNCTION_BLOCK MoveModuloTask EXTENDS TcoCore.TcoTask IMPLEMENTS ITcoDriveSimple
VAR
    {attribute addProperty Name "<#Position#>"}
    _position : LREAL;
    {attribute addProperty Name "<#Velocity#>"}
    _velocity : LREAL;
    {attribute addProperty Name "<#Acceleration#>"}
    _acceleration : LREAL;
    {attribute addProperty Name "<#Deceleration#>"}
    _deceleration : LREAL;
    {attribute addProperty Name "<#Jerk#>"}
    _jerk : LREAL;
    {attribute addProperty Name "<#Direction#>"}
    _direction : eDirection;
END_VAR
VAR
    {attribute 'hide'}
    _axisRef : REFERENCE TO TcoAxisRef;
    {attribute 'hide'}
    _mcMoveModulo : Tc2_MC2.MC_MoveModulo;
    {attribute 'hide'}
    _mc_direction : Tc2_MC2.MC_Direction;
    {attribute 'hide'}
    _message : STRING(125);
    {attribute 'hide'}
    _dummyPreconditionOK : BOOL;
END_VAR

IF NOT __ISVALIDREF(_axisRef) THEN
    IF __ISVALIDREF(DriveRef) THEN
        _axisRef REF= DriveRef.AxisRef;
    ELSE
        RETURN;
    END_IF
END_IF

IF Execute() THEN
    _dummyPreconditionOK := TRUE;

    IF NOT DriveRef._movementState.MovePreconditionsOk(THIS^, _dummyPreconditionOK) THEN
        Messenger.Error('To be implemented');
        RETURN;
    END_IF

    _mcMoveModulo(Axis := _axisRef,
        Execute := NOT _mcMoveModulo.Busy,
        Position := _position,
        Velocity := _velocity,
        Acceleration := _acceleration,
        Deceleration := _deceleration,
        Jerk := _jerk,
        Direction := _mc_direction,
        BufferMode := Tc2_MC2.MC_Aborting,
        Done =>,
        Busy =>,
        Active =>,
        CommandAborted =>,
        Error =>,
        ErrorID =>);

    IF _mcMoveModulo.CommandAborted THEN
        THIS^.Abort();
    END_IF

    DoneWhen(_mcMoveModulo.Done);
    ThrowWhen(_mcMoveModulo.Error);
END_IF

PROPERTY DriveRef : REFERENCE TO TcoDriveSimple
GET
VAR
    _drive : ITcoDriveSimple := 0;
END_VAR
IF __QUERYINTERFACE(THIS^.Parent, _drive) THEN
    DriveRef REF= _drive.DriveRef;
END_IF
END_GET
END_PROPERTY

METHOD PUBLIC FB_init : BOOL
VAR_INPUT
    bInitRetains : BOOL; // if TRUE, the retain variables are initialized (warm start / cold start)
    bInCopyCode : BOOL; // if TRUE, the instance afterwards gets moved into the copy code (online change)
    ParentObject : ITcoObject;
END_VAR
END_METHOD

METHOD INTERNAL InvokeWithParams : ITcoTaskStatus
VAR_INPUT
    inPosition : LREAL;
    inVelocity : LREAL;
    inAcceleration : LREAL;
    inDeceleration : LREAL;
    inJerk : LREAL;
    inDirection : eDirection;
END_VAR
_position := inPosition;
_velocity := inVelocity;
_acceleration := inAcceleration;
_deceleration := inDeceleration;
_jerk := inJerk;
_direction := inDirection;
InvokeWithParams := THIS^.Invoke();
END_METHOD

(*~
    <docu>
        <summary>
            Executes when task is aborted.
        </summary>
    </docu>
~*)
METHOD PROTECTED OnAbort
IF NOT __ISVALIDREF(_axisRef) THEN
    IF __ISVALIDREF(DriveRef) THEN
        _axisRef REF= DriveRef.AxisRef;
    ELSE
        RETURN;
    END_IF
END_IF

THIS^.DriveRef.Stop(-1, -1);
_mcMoveModulo(Axis := _axisRef, Execute := FALSE);
THIS^.DriveRef._movementState.Restore();
END_METHOD

(*~
    <docu>
        <summary>
            Executes when task reaches the ```Done``` state .
        </summary>
    </docu>
~*)
METHOD PROTECTED OnDone
_mcMoveModulo(Axis := _axisRef, Execute := FALSE);
THIS^.DriveRef._movementState.Restore();
END_METHOD

(*~
    <docu>
        <summary>
            Executes when task reaches the ```Error``` state.
            <para>
                Do not confuse with <see cref="PlcDocu.TcoCore.TcoTask.WhileError()"/>, that is called cyclically until '''Error''' state is left.
            </para>
        </summary>
    </docu>
~*)
METHOD PROTECTED OnError
THIS^.DriveRef._movementState.Restore();

IF NOT _axisRef.Status.Error THEN
    DriveRef.SetErrorID(DriveRef._moveModuloTask._mcMoveModulo.ErrorID);
END_IF

_mcMoveModulo(Axis := _axisRef, Execute := FALSE);
END_METHOD

METHOD PROTECTED OnStart
IF NOT Tco_TO_Tc2MC2_Direction(_direction, _mc_direction) THEN
    _message := Tc2_Standard.CONCAT('Unable to cast _direction variable of type TcoDrivesBeckhoff.eDirection (', TO_STRING(_mc_direction));
    _message := Tc2_Standard.CONCAT(_message, ') to the type Tc2_MC2.MC_Direction!!!');
    THIS^.Messenger.Post(_message, TcoCore.eMessageCategory.ProgrammingError);
    ThrowWhen(TRUE);
    RETURN;
END_IF

_mcMoveModulo(Axis := _axisRef, Execute := FALSE);
END_METHOD

(*~
    <docu>
        <summary>
            Restores this instance to the Ready state. Can be called explicitly or from within one of the restore mechanisms.
            <para>
                See also <see cref="PlcDocu.TcoCore.TcoTask.AutoRestorable()"/>
            </para>
        </summary>
    </docu>
~*)
METHOD Restore : ITcoRestorable
SUPER^.Restore();
END_METHOD

(*~
    <docu>
        <summary>
            Executes until task is in ```Error``` state .
        </summary>
    </docu>
~*)
METHOD PROTECTED WhileError
IF NOT _axisRef.Status.Error THEN
    DriveRef.SetErrorID(DriveRef._moveModuloTask._mcMoveModulo.ErrorID);
    _mcMoveModulo(Axis := _axisRef, Execute := FALSE);
END_IF
END_METHOD

END_FUNCTION_BLOCK

// ---- POUs/Prototypes/CartesianCoordinateSystem/TcoAxisExchangeDataTask.TcPOU
(*~
    <docu>
        <summary>
            TcoAxisExchangeDataTask task is a remote task  <see cref="PlcDocu.TcoCore.RemoteTask"/> with a paramater.
        </summary>
        <param name="_identifier">The Identifier, ID  of an entity on which a CRUD operation should be executed</param>
        <remarks>Inxton is required for this feature to work</remarks>
    </docu>
~*)
FUNCTION_BLOCK TcoAxisExchangeDataTask EXTENDS TcoCore.TcoRemoteTask
VAR
    (*~
    <docu>
        <summary>
            The Identifier, ID  of an entity on which a CRUD operation should be executed.
        </summary>
    </docu>
    ~*)
    _identifier : STRING(255);
    _doesNotExist : BOOL;
    _exchangeSuccessfuly : BOOL;
END_VAR

SUPER^();

PROPERTY PUBLIC DoesNotExist : bool
GET
DoesNotExist := _doesNotExist;
END_GET
END_PROPERTY

PROPERTY ReadSuccessfuly : bool
GET
ReadSuccessfuly := _exchangeSuccessfuly;
END_GET
END_PROPERTY

(*~
    <docu>
        <summary>
            Restores this instance to the Ready state. Can be called explicitly or from within one of the restore mechanisms.
            <para>
                See also <see cref="PlcDocu.TcoCore.TcoTask.AutoRestorable()"/>
            </para>
        </summary>
    </docu>
~*)
METHOD Restore : ITcoRestorable
VAR
END_VAR
_doesNotExist := FALSE;
//_identifier:='';
_exchangeSuccessfuly := FALSE;
SUPER^.Restore();
END_METHOD

METHOD WithId : REFERENCE TO TcoAxisExchangeDataTask
VAR_INPUT
    (*~
    <docu>
        <summary>
            The Identifier, ID  of an entity on which a CRUD operation should be executed.
        </summary>
    </docu>
    ~*)
    inIdentifier : STRING(254);
END_VAR
THIS^._identifier := inIdentifier;
WithId REF= THIS^;
THIS^.Messenger.Build().Append('<#Loading/saving data item with id:#> ').Append(_identifier).As().AsTrace();
END_METHOD

END_FUNCTION_BLOCK

// ---- POUs/Prototypes/CartesianCoordinateSystem/SingleAxisSystem/TcoSingleAxis.TcPOU
FUNCTION_BLOCK TcoSingleAxis EXTENDS TcoCore.TcoComponent IMPLEMENTS ITcoSingleAxis
VAR_INPUT
    inEnable : BOOL;
    inEnablePositive : BOOL;
    inEnableNegative : BOOL;
    inCalibrationCam : BOOL;
    refAxis : REFERENCE TO TcoAxisRef;
END_VAR
VAR_IN_OUT
    inoPositions : TcoSingleAxisPositionsRootContainer;
END_VAR
VAR
    {attribute 'hide'}
    _axisRef : REFERENCE TO TcoAxisRef;
    {attribute addProperty Name "<#Axis#>"}
    _axis : TcoDriveSimple(THIS^);
    {attribute addProperty Name "<#Load positions Task#>"}
    _loadPositionTask : TcoAxisExchangeDataTask(THIS^);
    {attribute addProperty Name "<#Save positions Task#>"}
    _savePositionTask : TcoAxisExchangeDataTask(THIS^);
    {attribute addProperty Name "<#Positions#>"}
    {attribute clr [MemberByIdentity()]}
    _positions : TcoSingleAxisPositionsRootContainer(THIS^);
    {attribute addProperty Name "<#Move absolute Task#>"}
    _moveAbsoluteTask : TcoCore.TcoTask(THIS^);
    {attribute addProperty Name "<#Move relative Task#>"}
    _moveRelativeTask : TcoCore.TcoTask(THIS^);
    {attribute addProperty Name "<#Restore Task#>"}
    _restoreTask : TcoCore.TcoTask(THIS^);
    {attribute addProperty Name "<#Status#>"}
    {attribute clr [ReadOnly()]}
    _status : TcoSingleAxisStatus;
    {attribute addProperty Name "<#Config#>"}
    _config : TcoSingleAxisConfig;
    _moveParams : TcoSingleAxisMoveParam;
    {attribute 'hide'}
    _infoTimer : TON;
    {attribute 'hide'}
    _errorTimer : TON;
END_VAR

_positions := inoPositions;

IF NOT __ISVALIDREF(refAxis) THEN
    Messenger.Post('<#Invalid reference axis #>', TcoCore.eMessageCategory.ProgrammingError);
    RETURN;
END_IF

_axisRef REF= refAxis;
_savePositionTask();
_loadPositionTask();

_axis(inEnable := inEnable,
    inEnablePositive := inEnablePositive,
    inEnableNegative := inEnableNegative,
    inCalibrationCam := inCalibrationCam,
    inoAxisRef := _axisRef);
//*************MOVE ABSOLUTE********************
_moveAbsoluteTask.Enabled := NOT _moveRelativeTask.Busy;

IF _moveAbsoluteTask.Execute() THEN
    THIS^._axis.MoveAbsolute(inPosition := _moveParams.Position,
        inVelocity := _moveParams.Velocity,
        inAcceleration := _moveParams.Acceleration,
        inDeceleration := _moveParams.Deceleration,
        inJerk := _moveParams.Jerk);

    _moveAbsoluteTask.DoneWhen(THIS^._axis.MoveAbsoluteTask.Done);
    _moveAbsoluteTask.ThrowWhen(THIS^._axis.MoveAbsoluteTask.Error);
END_IF;
//****************************************
//*************MOVE RELATIVE********************
_moveRelativeTask.Enabled := NOT _moveAbsoluteTask.Busy;

IF _moveRelativeTask.Execute() THEN
    THIS^._axis.MoveRelative(inDistance := _moveParams.Position,
        inVelocity := _moveParams.Velocity,
        inAcceleration := _moveParams.Acceleration,
        inDeceleration := _moveParams.Deceleration,
        inJerk := _moveParams.Jerk);

    _moveRelativeTask.DoneWhen(THIS^._axis.MoveRelativeTask.Done);
    _moveRelativeTask.ThrowWhen(_errorTimer.Q OR THIS^._axis.MoveRelativeTask.Error);
END_IF;
//****************************************
//*************RESTORE********************
_restoreTask.Enabled := TRUE;

IF _restoreTask.Execute() THEN
    Restore();
END_IF
//****************************************
inoPositions := _positions;

PROPERTY Axis : REFERENCE TO TcoDriveSimple
GET
Axis REF= _axis;
END_GET
END_PROPERTY

METHOD CallTimers
VAR_INPUT
    inValue : BOOL;
END_VAR
IF __ISVALIDREF(Config) THEN
    _infoTimer(IN := inValue, PT := THIS^.Config.InfoTime);
    _errorTimer(IN := inValue, PT := THIS^.Config.ErrorTime);
END_IF;
END_METHOD

(*~
    <docu>
        <summary>
            Gets the configuration of the Axis.
        </summary>
    </docu>
~*)
PROPERTY Config : REFERENCE TO TcoSingleAxisConfig
GET
Config REF= _config;
END_GET
END_PROPERTY

PROPERTY PUBLIC LoadPositionsTask : REFERENCE TO TcoAxisExchangeDataTask
GET
LoadPositionsTask REF= _loadPositionTask;
END_GET
END_PROPERTY

METHOD MoveAbsolute : ITcoTaskStatus
VAR_INPUT
    MoveParams : TcoSingleAxisMoveParam;
END_VAR
_moveParams := MoveParams;
MoveAbsolute := THIS^._moveAbsoluteTask.Invoke();
END_METHOD

PROPERTY PUBLIC MoveAbsoluteTask : REFERENCE TO TcoCore.TcoTask
GET
MoveAbsoluteTask REF= _moveAbsoluteTask;
END_GET
END_PROPERTY

METHOD MoveRelative : ITcoTaskStatus
VAR_INPUT
    MoveParams : TcoSingleAxisMoveParam;
END_VAR
_moveParams := MoveParams;
MoveRelative := THIS^._moveRelativeTask.Invoke();
END_METHOD

PROPERTY PUBLIC MoveRelativeTask : REFERENCE TO TcoCore.TcoTask
GET
MoveRelativeTask REF= _moveRelativeTask;
END_GET
END_PROPERTY

METHOD ResetDrive : TcoCore.ITcoTaskStatus
ResetDrive := THIS^.Axis.Reset();
END_METHOD

(*~
    <docu>
        <summary>
            Restores this instance to the Ready state. Can be called explicitly or from within one of the restore mechanisms.
        </summary>
    </docu>
~*)
METHOD Restore : ITcoRestorable
_axis.Restore();
_restoreTask.Restore();
_savePositionTask.Restore();
_loadPositionTask.Restore();
_moveAbsoluteTask.Restore();
_moveRelativeTask.Restore();
CallTimers(FALSE);
Messenger.UnPin();
END_METHOD

PROPERTY PUBLIC SavePositionsTask : REFERENCE TO TcoAxisExchangeDataTask
GET
SavePositionsTask REF= _savePositionTask;
END_GET
END_PROPERTY

METHOD PROTECTED ServiceMode
THIS^._axis.Service();
END_METHOD

METHOD SoeReset : TcoCore.ITcoTaskStatus
SoeReset := THIS^.Axis.SoEReset();
END_METHOD

(*~
    <docu>
        <summary>
            Gets the status of the Axis system.
        </summary>
    </docu>
~*)
PROPERTY Status : REFERENCE TO TcoSingleAxisStatus
GET
Status REF= _status;
END_GET
END_PROPERTY

END_FUNCTION_BLOCK

// ---- POUs/Prototypes/CartesianCoordinateSystem/SingleAxisSystem/TcoSingleAxisPositionsRootContainer.TcPOU
FUNCTION_BLOCK TcoSingleAxisPositionsRootContainer EXTENDS TcoCore.TcoObject
VAR_INPUT
END_VAR
VAR_OUTPUT
END_VAR
VAR
END_VAR

END_FUNCTION_BLOCK
